TYPE ST_AxisName :
STRUCT
  sName     : STRING(31);
  bValid    : BOOL;
END_STRUCT
END_TYPE

(* stored: Version 1.1.0.1, ProductVersion 3.1.4023.8
   DUT ST_AxisName: Id {b6f71290-de11-4889-a4ba-25916bf9a8c4} *)
